TYPE ST_Values :
STRUCT
	  {attribute 'Unit' := 'm/s'}
	  {attribute 'DisplayName' := 'Speed'}
	  Sensor1   : REAL;
	  {attribute 'Unit' := 'V'}
	  {attribute 'DisplayName' := 'Voltage'}
	  Sensor2	: DINT;
	  {attribute 'Unit' := 'A'}
	  {attribute 'DisplayName' := 'Current'}
	  Sensor3	: DINT;
END_STRUCT
END_TYPE

(* stored: Version 1.1.0.1, ProductVersion 3.1.4024.5
   DUT ST_Values: Id {ddce2c5e-11a3-4b4a-bc6c-fee7cd53eab6} *)
